FUNCTION_BLOCK xPPU_Stamp
VAR_INPUT
	i_error: POINTER TO ErrorManager;
	i_process: POINTER TO ProcessManager;
	i_state: POINTER TO StateTracker;
END_VAR
VAR
	m_stampParams: ParameterSet;
	m_subRes: EOperationResult;
END_VAR

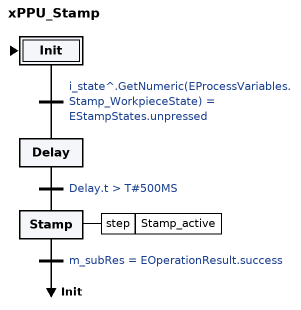
INITIAL_STEP Init:
END_STEP
TRANSITION FROM Init TO Delay
    := i_state^.GetNumeric(EProcessVariables.Stamp_WorkpieceState) = EStampStates.unpressed;
END_TRANSITION
STEP Delay:
END_STEP
TRANSITION FROM Delay TO Stamp
    := Delay.t > T#500MS;
END_TRANSITION
STEP Stamp:
    Stamp_active(N);  // step action
END_STEP
TRANSITION FROM Stamp TO Init
    := m_subRes = EOperationResult.success;
END_TRANSITION

ACTION Stamp_active:
m_stampParams.SetParam_Numeric('pressure_white', 4000);
m_stampParams.SetParam_Numeric('pressure_black', 4000);
m_stampParams.SetParam_Numeric('pressure_metal', 4000);

m_subRes := i_process^.Execute(
	EBehaviorType.control_primitive,
	EPrimitives.Stamp_StampWorkpiece,
	m_stampParams);
END_ACTION

END_FUNCTION_BLOCK

(* stored: Version 1.1.0.1, ProductVersion 3.1.4024.12
   POU xPPU_Stamp: Id {085d3a85-476d-4e64-b03f-4d0296436b8b}, SpecialFunc None
   Action Stamp_active: Id {2439002e-1d5d-496e-ad43-c117281d3379} *)
